Yaskawa INFORM job: LOAD_BOTTOM_START_XYZ.JBI

/JOB
//NAME LOAD_BOTTOM_START_XYZ
///FOLDERNAME FOLDER001
//POS
///NPOS 0,0,0,1,0,0
///TOOL 1
///POSTYPE ROBOT
///RECTAN
///RCONF 0,0,0,0,0,0,0,0,0,0,0,0,0,0,0,0,0,0,0,0,0,0,0,0
P00094=792.896,160.291,471.972,0.0813,10.0064,0.0684
//INST
///DATE 2025/09/26 17:01
///ATTR SC,RW
///GROUP1 RB1
NOP
'GET X Y Z VALUE FOR BOTTOM START
'X
GETE D073 P094 (1)
SET I073  EXPRESS I072 * 100
IFTHENEXP I073>10000
	 SET I073 10000
ELSEIFEXP I073<-10000
	 SET I073 -10000
ENDIF
'Y
GETE D075 P094 (2)
SET I075  EXPRESS I074 * 100
IFTHENEXP I075>10000
	 SET I075 10000
ELSEIFEXP I075<-10000
	 SET I075 -10000
ENDIF
'Z
GETE D077 P094 (3)
SET I077  EXPRESS I076 * 100
IFTHENEXP I077>10000
	 SET I077 10000
ELSEIFEXP I077<-10000
	 SET I077 -10000
ENDIF
'ADD THE CORRECTIONS
ADD D073 I073
SETE P094 (1) D073
ADD D075 I075
SETE P094 (2) D075
ADD D077 I077
SETE P094 (3) D077
'SET TO 0
SET I072 0
SET I073 0
SET I074 0
SET I075 0
SET I076 0
SET I077 0
END
